TYPE RouterMemory :
STRUCT
	startMemory : DINT;
	currentMemory : DINT;
	memoryDifference : DINT;
	tcStartMemory : DINT;
	tcStartMemoryDifference : DINT;
END_STRUCT
END_TYPE

(* stored: Version 1.1.0.1, ProductVersion 3.1.4024.12
   DUT RouterMemory: Id {33158f14-6646-0e3d-3fc0-b5120ef35cc6} *)
